FUNCTION_BLOCK PML_Method_Base
VAR_INPUT
END_VAR
VAR_OUTPUT
END_VAR
VAR
	ipackml : IPmlStateMachine;
END_VAR

METHOD PROTECTED Aborted : BOOL
VAR_INPUT
END_VAR
END_METHOD

METHOD PROTECTED Aborting : BOOL
VAR_INPUT
END_VAR
ipackml.SetStateComplete();
END_METHOD

METHOD PROTECTED Clearing : BOOL
VAR_INPUT
END_VAR
ipackml.SetStateComplete();
END_METHOD

METHOD PROTECTED Completed : BOOL
VAR_INPUT
END_VAR
END_METHOD

METHOD PROTECTED Completing : BOOL
VAR_INPUT
END_VAR
ipackml.SetStateComplete();
END_METHOD

METHOD PUBLIC Cycle : BOOL
VAR_INPUT
END_VAR
CASE ipackml.GetCurrentState() OF
	E_PMLState.ePMLState_Clearing:
		Clearing();
	E_PMLState.ePMLState_Aborted:
		Aborted();
	E_PMLState.ePMLState_Aborting:
		Aborting();
	E_PMLState.ePMLState_Complete:
		Completed();
	E_PMLState.ePMLState_Completing:
		Completing();
	E_PMLState.ePMLState_Execute:
		Execute();
	E_PMLState.ePMLState_Held:
		Held();
	E_PMLState.ePMLState_Holding:
		Holding();
	E_PMLState.ePMLState_Idle:
		Idle();
	E_PMLState.ePMLState_Resetting:
		Resetting();
	E_PMLState.ePMLState_Starting:
		Starting();
	E_PMLState.ePMLState_Stopped:
		Stopped();
	E_PMLState.ePMLState_Stopping:
		Stopping();
	E_PMLState.ePMLState_Suspended:
		Suspended();
	E_PMLState.ePMLState_Suspending:
		Suspending();
	E_PMLState.ePMLState_Undefined:
		Undefined();
	E_PMLState.ePMLState_Unholding:
		Unholding();
	E_PMLState.ePMLState_Unsuspending:
		Unsuspending();
END_CASE
END_METHOD

METHOD PROTECTED Execute : BOOL
VAR_INPUT
END_VAR
END_METHOD

METHOD PROTECTED Held : BOOL
VAR_INPUT
END_VAR
END_METHOD

METHOD PROTECTED Holding : BOOL
VAR_INPUT
END_VAR
ipackml.SetStateComplete();
END_METHOD

METHOD PROTECTED Idle : BOOL
VAR_INPUT
END_VAR
END_METHOD

PROPERTY PUBLIC PackMLStateMachine : IPmlStateMachine
GET
PackMLStateMachine := ipackml;
END_GET
SET
ipackml := PackMLStateMachine;
END_SET
END_PROPERTY

METHOD PROTECTED Resetting : BOOL
VAR_INPUT
END_VAR
ipackml.SetStateComplete();
END_METHOD

METHOD PROTECTED Starting : BOOL
VAR_INPUT
END_VAR
ipackml.SetStateComplete();
END_METHOD

METHOD PROTECTED Stopped : BOOL
VAR_INPUT
END_VAR
END_METHOD

METHOD PROTECTED Stopping : BOOL
VAR_INPUT
END_VAR
ipackml.SetStateComplete();
END_METHOD

METHOD PROTECTED Suspended : BOOL
VAR_INPUT
END_VAR
END_METHOD

METHOD PROTECTED Suspending : BOOL
VAR_INPUT
END_VAR
ipackml.SetStateComplete();
END_METHOD

METHOD PROTECTED Undefined : BOOL
VAR_INPUT
END_VAR
END_METHOD

METHOD PROTECTED Unholding : BOOL
VAR_INPUT
END_VAR
ipackml.SetStateComplete();
END_METHOD

METHOD PROTECTED Unsuspending : BOOL
VAR_INPUT
END_VAR
ipackml.SetStateComplete();
END_METHOD

END_FUNCTION_BLOCK

(* stored: Version 1.1.0.1, ProductVersion 3.1.4024.12
   POU PML_Method_Base: Id {a3013dfd-707d-4828-8b6c-b9533715f53c}, SpecialFunc None
   Folder Action_States: Id {ed13041c-08c9-43cf-86f5-29ff88150424}
   Folder Wait_States: Id {b8022189-ff74-4d04-ae1f-588844f6f7ac}
   Method Aborted: Id {2ebbd337-bec1-4af5-b3d2-47f5b1b4bb08}
   Method Aborting: Id {8ebfbf21-c6a5-403c-9487-ff796f1db8e7}
   Method Clearing: Id {56493295-8f17-451f-bb25-1c47b8aaecda}
   Method Completed: Id {0aa614b6-c84f-4ba8-a564-142a8c1cec68}
   Method Completing: Id {a51b2a5d-7442-44cf-a70e-11b8597d7104}
   Method Cycle: Id {1df90c6e-7792-4f54-826d-f960e9e1aaf2}
   Method Execute: Id {04ce3673-8ac1-4eec-b2ae-c3f3a53c95cd}
   Method Held: Id {5514a7a2-0379-4d20-bcb7-31007c04498a}
   Method Holding: Id {487c6d80-7ce0-49ec-90da-146a8e6cbb35}
   Method Idle: Id {99adc4a5-311c-4e5b-bc06-7c2ffd3aaf3f}
   Property PackMLStateMachine: Id {c16aaacf-fd3a-443a-85a5-b963678c1753}
   Get Get: Id {d66b1fe6-46f7-4342-8172-35648ad321b3}
   Set Set: Id {c8eef4aa-d747-4773-817f-54fc663564f7}
   Method Resetting: Id {ab086979-824f-4e2d-9086-0949108db333}
   Method Starting: Id {b834ab70-1436-4b93-baf6-26fb7bdadd6e}
   Method Stopped: Id {786f468a-9460-4066-ae27-dd538204f76f}
   Method Stopping: Id {06b02fb1-cb5e-4932-9d1c-cdb86d08d66c}
   Method Suspended: Id {5c9c15f9-3566-49ce-b6a1-ef9fc1ef3868}
   Method Suspending: Id {83a174bb-dddc-4533-ad7b-e3097df8a6a1}
   Method Undefined: Id {7c81348a-df94-4779-8c3e-bf626771acbb}
   Method Unholding: Id {09d74fc9-52b4-42e6-9217-c802ab62da32}
   Method Unsuspending: Id {f4d8b750-db5e-489f-9b33-bbf870c76a22} *)
